Staubli VAL3: AtHome.pgx

public program AtHome(bool x_bHome (dimensions=1))
begin


  dDio["O1_bFollowDone"]=x_bHome
  call Digtal2Analog()







end
